// Mitsubishi GX Works2 project: 互锁以及触发   PLC: Q13UDV

// global labels: Global1
VAR_GLOBAL
  xbpos : ARRAY [1..4] OF BOOL;
  ybpos : ARRAY [1..4] OF BOOL;
  zbpos : ARRAY [1..4] OF BOOL;
END_VAR

PROGRAM 主程序
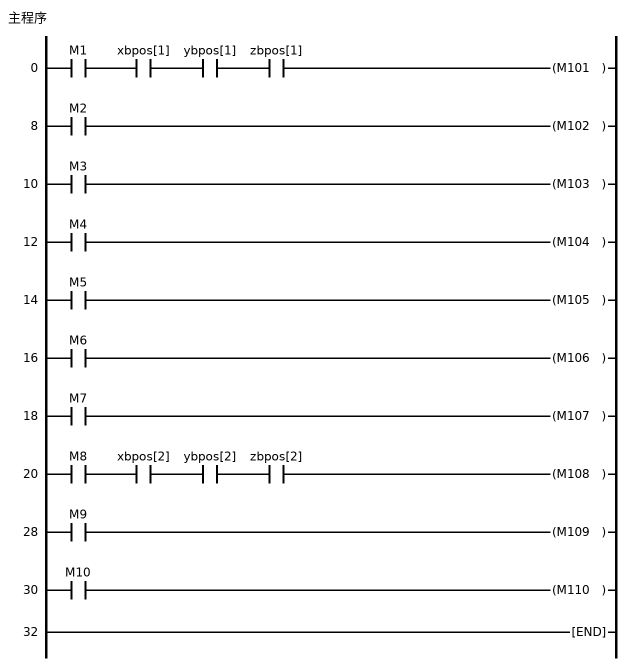
0     LD      M1
      AND     xbpos[1]
      AND     ybpos[1]
      AND     zbpos[1]
      OUT     M101
8     LD      M2
      OUT     M102
10    LD      M3
      OUT     M103
12    LD      M4
      OUT     M104
14    LD      M5
      OUT     M105
16    LD      M6
      OUT     M106
18    LD      M7
      OUT     M107
20    LD      M8
      AND     xbpos[2]
      AND     ybpos[2]
      AND     zbpos[2]
      OUT     M108
28    LD      M9
      OUT     M109
30    LD      M10
      OUT     M110
32    END
END_PROGRAM

PROGRAM 中间互锁
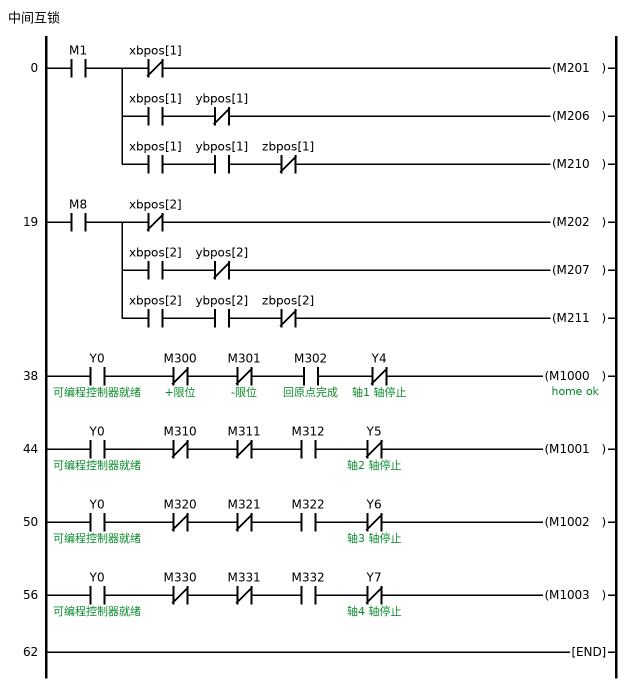
0     LD      M1
      MPS
      ANI     xbpos[1]
      OUT     M201
      MRD
      AND     xbpos[1]
      ANI     ybpos[1]
      OUT     M206
      MPP
      AND     xbpos[1]
      AND     ybpos[1]
      ANI     zbpos[1]
      OUT     M210
19    LD      M8
      MPS
      ANI     xbpos[2]
      OUT     M202
      MRD
      AND     xbpos[2]
      ANI     ybpos[2]
      OUT     M207
      MPP
      AND     xbpos[2]
      AND     ybpos[2]
      ANI     zbpos[2]
      OUT     M211
38    LD      Y0  ; 可编程控制器就绪
      ANI     M300  ; +限位
      ANI     M301  ; -限位
      AND     M302  ; 回原点完成
      ANI     Y4  ; 轴1 轴停止
      OUT     M1000  ; home ok
44    LD      Y0  ; 可编程控制器就绪
      ANI     M310
      ANI     M311
      AND     M312
      ANI     Y5  ; 轴2 轴停止
      OUT     M1001
50    LD      Y0  ; 可编程控制器就绪
      ANI     M320
      ANI     M321
      AND     M322
      ANI     Y6  ; 轴3 轴停止
      OUT     M1002
56    LD      Y0  ; 可编程控制器就绪
      ANI     M330
      ANI     M331
      AND     M332
      ANI     Y7  ; 轴4 轴停止
      OUT     M1003
62    END
END_PROGRAM

PROGRAM 触发
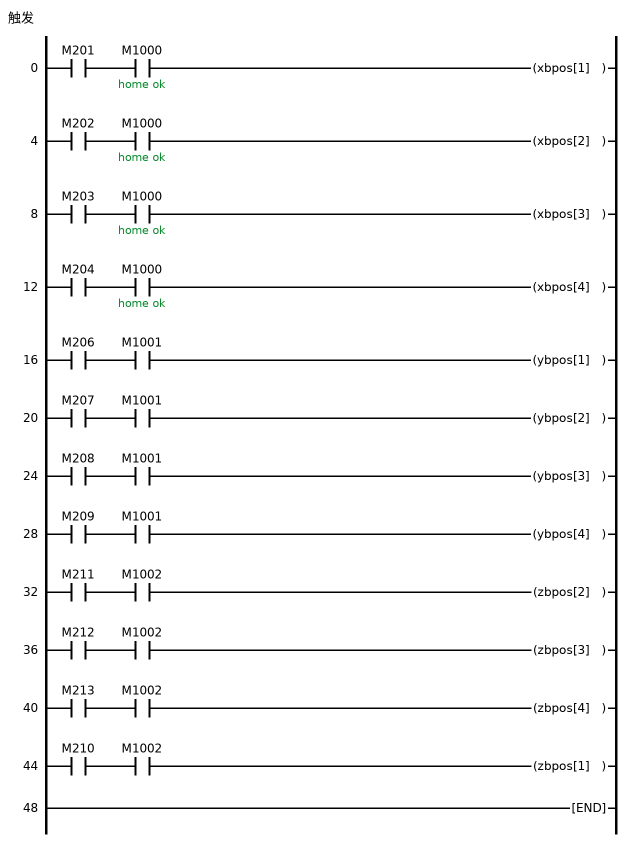
0     LD      M201
      AND     M1000  ; home ok
      OUT     xbpos[1]
4     LD      M202
      AND     M1000  ; home ok
      OUT     xbpos[2]
8     LD      M203
      AND     M1000  ; home ok
      OUT     xbpos[3]
12    LD      M204
      AND     M1000  ; home ok
      OUT     xbpos[4]
16    LD      M206
      AND     M1001
      OUT     ybpos[1]
20    LD      M207
      AND     M1001
      OUT     ybpos[2]
24    LD      M208
      AND     M1001
      OUT     ybpos[3]
28    LD      M209
      AND     M1001
      OUT     ybpos[4]
32    LD      M211
      AND     M1002
      OUT     zbpos[2]
36    LD      M212
      AND     M1002
      OUT     zbpos[3]
40    LD      M213
      AND     M1002
      OUT     zbpos[4]
44    LD      M210
      AND     M1002
      OUT     zbpos[1]
48    END
END_PROGRAM

// device comments not shown above
X0  ; QD75准备完成
X1  ; 同步用标记
X4  ; 轴1 M代码ON
X5  ; 轴2 M代码ON
X6  ; 轴3 M代码ON
X7  ; 轴4 M代码ON
X8  ; 轴1 错误检测
X9  ; 轴2 错误检测
X0A  ; 轴3 错误检测
X0B  ; 轴4 错误检测
X0C  ; 轴1 BUSY
X0D  ; 轴2 BUSY
X0E  ; 轴3 BUSY
X0F  ; 轴4 BUSY
X10  ; 轴1 启动完成
X11  ; 轴2 启动完成
X12  ; 轴3 启动完成
X13  ; 轴4 启动完成
X14  ; 轴1 定位完成
X15  ; 轴2 定位完成
X16  ; 轴3 定位完成
X17  ; 轴4 定位完成
Y8  ; 轴1 正转JOG启动
Y9  ; 轴1 反转JOG启动
Y0A  ; 轴2 正转JOG启动
Y0B  ; 轴2 反转JOG启动
Y0C  ; 轴3 正转JOG启动
Y0D  ; 轴3 反转JOG启动
Y0E  ; 轴4 正转JOG启动
Y0F  ; 轴4 反转JOG启动
Y10  ; 轴1 定位启动
Y11  ; 轴2 定位启动
Y12  ; 轴3 定位启动
Y13  ; 轴4 定位启动
Y14  ; 轴1 执行禁止标记
Y15  ; 轴2 执行禁止标记
Y16  ; 轴3 执行禁止标记
Y17  ; 轴4 执行禁止标记
